FUNCTION_BLOCK EMERGENCY_CONTROLLER (* Composite Function Block Type *)
  (* Standard: 61499-2 *)
  (* Version 1.0, 2019-03-16, adeel *)
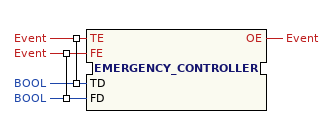
  EVENT_INPUT
    TE WITH TD; (* Initialization Request *)
    FE WITH FD; (* Normal Execution Request *)
  END_EVENT
  EVENT_OUTPUT
    OE; (* Initialization Confirm *)
  END_EVENT
  VAR_INPUT
    TD : BOOL; (* Input event qualifier *)
    FD : BOOL;
  END_VAR
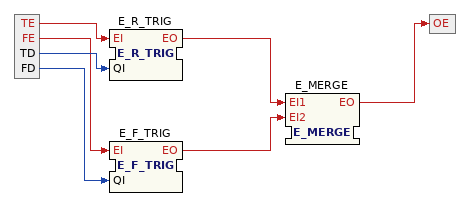
  FBS
    E_F_TRIG : E_F_TRIG;
    E_R_TRIG : E_R_TRIG;
    E_MERGE : E_MERGE;
  END_FBS
  EVENT_CONNECTIONS
    TE TO E_R_TRIG.EI;
    FE TO E_F_TRIG.EI;
    E_R_TRIG.EO TO E_MERGE.EI1;
    E_F_TRIG.EO TO E_MERGE.EI2;
    E_MERGE.EO TO OE;
  END_CONNECTIONS
  DATA_CONNECTIONS
    TD TO E_R_TRIG.QI;
    FD TO E_F_TRIG.QI;
  END_CONNECTIONS
END_FUNCTION_BLOCK
